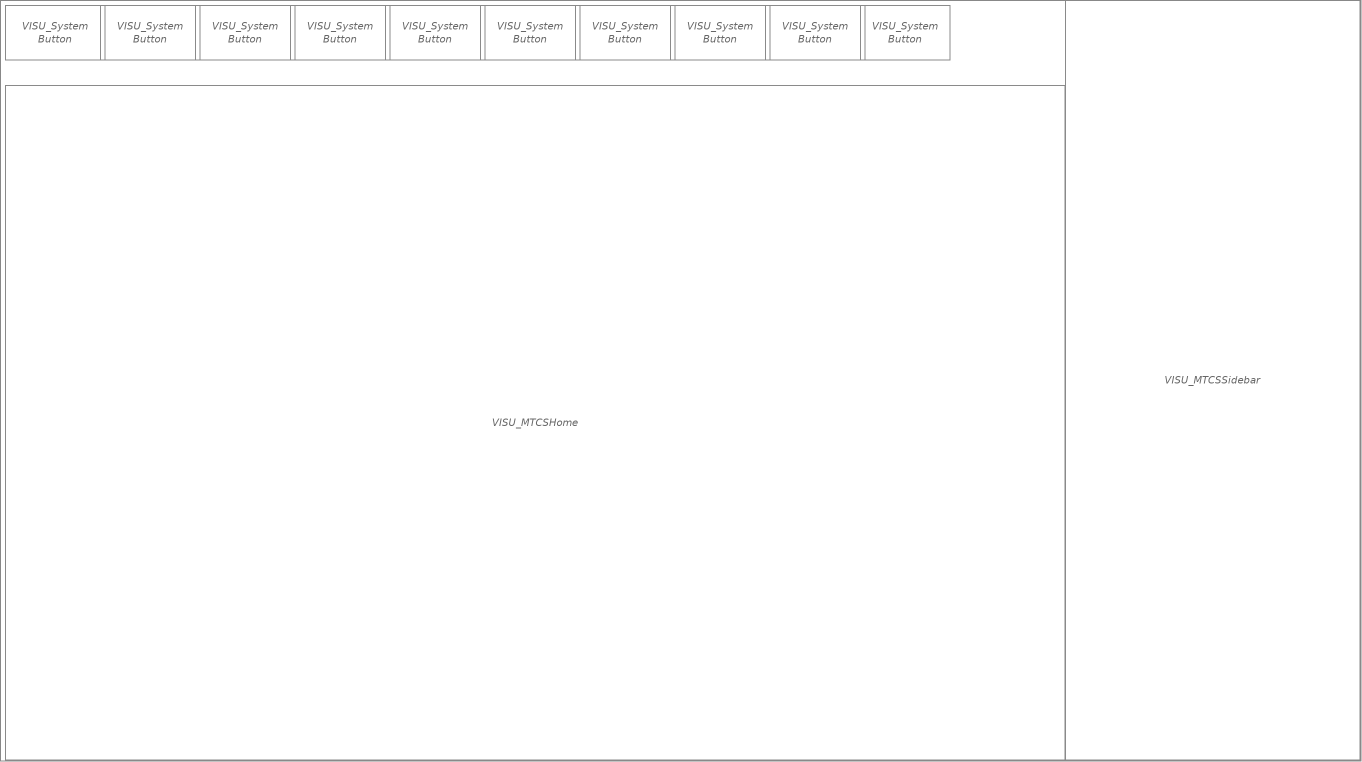
VISUALIZATION VISU_MTCS  // 1362x762
VAR_IN_OUT
	mtcs : MTCS;
	mtcsWidget : MTCSWidget;
END_VAR
    Frame (5,85 1060x675)
        shows VISU_MTCSHome(mtcs := mtcs, mtcsWidget := mtcsWidget)
        shows VISU_Services(ref := mtcs.parts.services, widget := mtcsWidget.services)
        shows VISU_Cover(ref := mtcs.parts.cover, widget := mtcsWidget.cover)
        shows VISU_M1(ref := mtcs.parts.m1, widget := mtcsWidget.m1)
        shows VISU_M2(ref := mtcs.parts.m2, ref_io := mtcs.parts.m1.parts.io, widget := mtcsWidget.m2)
        shows VISU_M3(m3 := mtcs.parts.m3, m3Widget := mtcsWidget.m3)
        shows VISU_Telemetry(ref := mtcs.parts.telemetry, widget := mtcsWidget.telemetry)
        shows VISU_Hydraulics(ref := mtcs.parts.hydraulics, widget := mtcsWidget.hydraulics, ref_safetyHydraulics := mtcs.parts.safety.parts.hydraulics, ref_safetyIO := mtcs.parts.safety.parts.io)
        shows VISU_Safety(ref := mtcs.parts.safety, widget := mtcsWidget.safety)
        shows VISU_Axes(ref := mtcs.parts.axes, widget := mtcsWidget.axes)
        p3520207131: GVL.mtcsWidget.m3
        p2783583907: mtcs.parts.m1.parts.io
        p446882865: mtcs.parts.services
        p3849118168: mtcsWidget.services
    Frame (5,5 100x55)
        shows VISU_SystemButton(widget := mtcsWidget.button_home)
        OnMouseClick: FrameSelectionChange Selection=SelectedFrame=eff586ae-9280-4d77-af51-f88c6c7c4d0e, GlobSel=AssignType=Directly, SelType=Locally
        OnMouseClick: execute { mtcsWidget.activeTab := MTCSTabs.HOME; }
    Frame (195,5 100x55)
        shows VISU_SystemButton(widget := mtcsWidget.button_cover)
        OnMouseClick: FrameSelectionChange Selection=SelectedFrame=eff586ae-9280-4d77-af51-f88c6c7c4d0e, Selection=2, GlobSel=AssignType=Directly, SelType=Locally
        OnMouseClick: execute { mtcsWidget.activeTab := MTCSTabs.COVER; }
    Frame (1065,0 295x760)
        shows VISU_MTCSSidebar(mtcs := mtcs, mtcsWidget := mtcsWidget)
    Frame (290,5 100x55)
        shows VISU_SystemButton(widget := mtcsWidget.button_m1)
        OnMouseClick: FrameSelectionChange Selection=SelectedFrame=eff586ae-9280-4d77-af51-f88c6c7c4d0e, Selection=3, GlobSel=AssignType=Directly, SelType=Locally
        OnMouseClick: execute { mtcsWidget.activeTab := MTCSTabs.M1; }
    Frame (480,5 100x55)
        shows VISU_SystemButton(widget := mtcsWidget.button_m3)
        OnMouseClick: FrameSelectionChange Selection=SelectedFrame=eff586ae-9280-4d77-af51-f88c6c7c4d0e, Selection=5, GlobSel=AssignType=Directly, SelType=Locally
        OnMouseClick: execute { mtcsWidget.activeTab := MTCSTabs.M3; }
    Frame (100,5 100x55)
        shows VISU_SystemButton(widget := mtcsWidget.button_services)
        OnMouseClick: FrameSelectionChange Selection=SelectedFrame=eff586ae-9280-4d77-af51-f88c6c7c4d0e, Selection=1, GlobSel=AssignType=Directly, SelType=Locally
        OnMouseClick: execute { mtcsWidget.activeTab := MTCSTabs.SERVICES; }
    Frame (575,5 100x55)
        shows VISU_SystemButton(widget := mtcsWidget.button_telemetry)
        OnMouseClick: FrameSelectionChange Selection=SelectedFrame=eff586ae-9280-4d77-af51-f88c6c7c4d0e, Selection=6, GlobSel=AssignType=Directly, SelType=Locally
        OnMouseClick: execute { mtcsWidget.activeTab := MTCSTabs.TELEMETRY; }
    Frame (385,5 100x55)
        shows VISU_SystemButton(widget := mtcsWidget.button_m2)
        OnMouseClick: FrameSelectionChange Selection=SelectedFrame=eff586ae-9280-4d77-af51-f88c6c7c4d0e, Selection=4, GlobSel=AssignType=Directly, SelType=Locally
        OnMouseClick: execute { mtcsWidget.activeTab := MTCSTabs.M2; }
    Frame (670,5 100x55)
        shows VISU_SystemButton(widget := mtcsWidget.button_hydraulics)
        OnMouseClick: FrameSelectionChange Selection=SelectedFrame=eff586ae-9280-4d77-af51-f88c6c7c4d0e, Selection=7, GlobSel=AssignType=Directly, SelType=Locally
        OnMouseClick: execute { mtcsWidget.activeTab := MTCSTabs.HYDRAULICS; }
    Frame (765,5 100x55)
        shows VISU_SystemButton(widget := mtcsWidget.button_safety)
        OnMouseClick: FrameSelectionChange Selection=SelectedFrame=eff586ae-9280-4d77-af51-f88c6c7c4d0e, Selection=8, GlobSel=AssignType=Directly, SelType=Locally
        OnMouseClick: execute { mtcsWidget.activeTab := MTCSTabs.SAFETY; }
    Frame (860,5 90x55)
        shows VISU_SystemButton(widget := mtcsWidget.button_axes)
        OnMouseClick: FrameSelectionChange Selection=SelectedFrame=eff586ae-9280-4d77-af51-f88c6c7c4d0e, Selection=9, GlobSel=AssignType=Directly, SelType=Locally
        OnMouseClick: execute { mtcsWidget.activeTab := MTCSTabs.AXES; }
END_VISUALIZATION

(* stored: Version 1.1.0.1, ProductVersion 3.1.4019.2
   Visu VISU_MTCS: Id {0d2db229-d8d9-49d0-9c41-25d723d71f45} *)
